TYPE DUT_TASKSTATE :
(
	Unassigned := 0,
	Assigned := 1,
	WaitingForSkillReady := 2,
	InProgress := 3,
	Done := 4,
	Aborted := 5,
	Error := 6
);
END_TYPE

(* stored: Version 1.1.0.1, ProductVersion 3.1.0.25
   DUT DUT_TASKSTATE: Id {37fc6dab-3950-4b72-9da5-f33a5868748f} *)
